FUNCTION_BLOCK FB_FileWriter
VAR_INPUT
	sFilePath					: T_MaxString; 
	sFileName					: T_MaxString;
	sNetId						: STRING; // NetId of the target, leave empty for local
END_VAR
VAR CONSTANT
	nArrBufferSize				: INT := 1000; 	
END_VAR
VAR
    fbFileOpen  				: FB_FileOpen;
    fbFilePuts  				: FB_FilePuts;
    fbFileClose 				: FB_FileClose;
    nFileHandle 				: UINT;
	
    arrBuffer   				: ARRAY[0..nArrBufferSize] OF T_MaxString;
    eFileWriteState 			: (IDLE, OPEN_FILE, WRITE_TO_FILE, CLOSE_FILE, ERROR);
END_VAR

CASE eFileWriteState OF
    IDLE:
        // Make sure all the file writing FBs are ready for use (trigger on execute)
        Init();
        
        // We have pending data to be written
        IF arrBuffer[0] <> '' THEN // Makes sure that the first element of the array is not an empty string 
            eFileWriteState := OPEN_FILE;
        END_IF
        
    OPEN_FILE:
        // Opens a file for writing at the end of the file (append). 
        // If the file does not exist, a new file is created.
        fbFileOpen(
            bExecute    := TRUE,
            sNetId      := sNetId,
            sPathName   := CONCAT(sFilePath, sFileName),
            nMode       := FOPEN_MODEAPPEND);
            
        IF fbFileOpen.bError THEN
            eFileWriteState := ERROR;
        ELSIF NOT fbFileOpen.bBusy THEN
            nFileHandle := fbFileOpen.hFile;
            fbFileOpen(bExecute := FALSE);
            eFileWriteState := WRITE_TO_FILE;
        END_IF
    
    WRITE_TO_FILE:
        fbFilePuts(
            bExecute    := TRUE,
            sNetId      := sNetId,
            hFile       := nFileHandle,
            sLine       := arrBuffer[0]); // Write the first element of the buffer
        
        IF fbFilePuts.bError THEN
            eFileWriteState := ERROR;
        ELSIF NOT fbFilePuts.bBusy THEN
            fbFilePuts(bExecute := FALSE);
            RotateBuffer(); // Remove the written data from the buffer
            eFileWriteState := CLOSE_FILE;
        END_IF
    
    CLOSE_FILE:
        fbFileClose(
            bExecute := TRUE,
            sNetId      := sNetId,
            hFile       := nFileHandle);
            
        IF fbFileClose.bError THEN
            eFileWriteState := ERROR;
        ELSIF NOT fbFileClose.bBusy THEN
            nFileHandle := 0;
            eFileWriteState := IDLE;
        END_IF      
    
    ERROR:
        // Error, clear the handle and go back to idle
        nFileHandle := 0;
        eFileWriteState := IDLE;
END_CASE

PROPERTY PUBLIC FileWriteState : STRING
GET
CASE eFileWriteState OF
    IDLE: 
        FileWriteState := 'IDLE';
    OPEN_FILE: 
        FileWriteState := 'OPEN_FILE';
    WRITE_TO_FILE: 
        FileWriteState := 'WRITE_TO_FILE';
    CLOSE_FILE: 
        FileWriteState := 'CLOSE_FILE';
    ERROR: 
        FileWriteState := 'ERROR';
ELSE
    FileWriteState := 'UNKNOWN';
END_CASE
END_GET
END_PROPERTY

METHOD PRIVATE Init
fbFileClose(bExecute := FALSE);
fbFileOpen(bExecute := FALSE);
fbFilePuts(bExecute := FALSE);
END_METHOD

METHOD PRIVATE InsertToBuffer 
VAR_INPUT
	value					: STRING;
END_VAR
VAR
    nBufferIndex    : INT;
END_VAR
FOR nBufferIndex := 0 TO nArrBufferSize BY 1 DO
    IF arrBuffer[nBufferIndex] = '' THEN
        // We found the free spot in the buffer, insert the value to this place
        arrBuffer[nBufferIndex] := value;
        EXIT;
    END_IF
END_FOR
END_METHOD

METHOD PRIVATE RotateBuffer

VAR
    nIndex  : int := 0;
END_VAR
FOR nIndex := 0 TO nArrBufferSize - 1 BY 1 DO
    // We can exit when we reached the empty slot in the buffer
    IF arrBuffer[nIndex] = '' THEN
        EXIT;
    END_IF
    // FIFO, removing first element in the array copying the next, etc...
    arrBuffer[nIndex] := arrBuffer[nIndex+1];
END_FOR
arrBuffer[nArrBufferSize-1] := ''; // Clear the last element after rotation
END_METHOD

METHOD PUBLIC WriteToFile
VAR_INPUT
    message : T_MaxString;
END_VAR
InsertToBuffer(value := message);
END_METHOD

END_FUNCTION_BLOCK

(* stored: Version 1.1.0.1, ProductVersion 3.1.4024.12
   POU FB_FileWriter: Id {7ec5e9a7-2d10-4582-aa4f-c19345b5de2f}, SpecialFunc None
   Property FileWriteState: Id {a921f34b-1325-4092-9bb6-f04add859cbc}
   Get Get: Id {60b04697-2267-4456-9987-9daa8ed392d7}
   Method Init: Id {eefdbfeb-6de0-4c9e-bca7-3ada7faf4662}
   Method InsertToBuffer: Id {d1cc2012-e617-4228-a52f-ddcc22d6a63d}
   Method RotateBuffer: Id {d626922d-400b-49f2-9da6-174abcfd43e4}
   Method WriteToFile: Id {06c32fea-3236-491d-81ca-2ba3d41d947c} *)
